(* Logix 5000 project; controller Savage_Saw vendor 1 type 14 code 154 rev 37.11; software revision 37.01; part 2 of 3 *)
(* tags used below, declared in another part *)
   AnyJogRise : BOOL;
   AnyJogStorage : BOOL;
   iAxis : DINT;
   ManualSpinCCW : BOOL;
   ManualSpinCW : BOOL;
   spinActive : BOOL;
   spinDemand : BOOL;
   timerSpinDownCCW : TIMER;
   timerSpinDownCW : TIMER;
   Auto : BOOL;
   AutoCutCancel : BOOL;
   AutoCutCancelFall : BOOL;
   AutoCutCancelOSF : BOOL;
   AutoCutReq : BOOL;
   AutoCutStartONS : BOOL;
   AutoCutStateChange : BOOL;
   AutoSpinCCW : BOOL;
   AutoSpinCW : BOOL;
   Axis : AxisData[3];
   AxisX_Gauge : ALIAS FOR Axis[0];
   AxisY_Traverse : ALIAS FOR Axis[1];
   AxisZ_RaiseLower : ALIAS FOR Axis[2];
   BladeChange10 : BOOL;
   BladeChange10ONS : BOOL;
   BladeChange20 : BOOL;
   BladeChange20ONS : BOOL;
   BladeChangeDone : BOOL;
   BladeChangeStartONS : BOOL;
   BladeChangeStateChange : BOOL;
   BladeMeasure10ONS : BOOL;
   BladeMeasure10StopAll : BOOL;
   BladeMeasure15ClearZero : BOOL;
   BladeMeasure20ONS : BOOL;
   BladeMeasure20Retract : BOOL;
   BladeMeasure30ONS : BOOL;
   BladeMeasure30Traverse : BOOL;
   BladeMeasure40Lower : BOOL;
   BladeMeasure40ONS : BOOL;
   BladeMeasure50ONS : BOOL;
   BladeMeasure50Stop : BOOL;
   BladeMeasure55ONS : BOOL;
   BladeMeasure55Raise : BOOL;
   BladeMeasure60ONS : BOOL;
   BladeMeasure60Stop : BOOL;
   BladeMeasure65Measure : BOOL;
   BladeMeasure65ONS : BOOL;
   BladeMeasure70Calc : BOOL;
   BladeMeasure70ONS : BOOL;
   BladeMeasure75ONS : BOOL;
   BladeMeasure75PartRef : BOOL;
   BladeMeasure80ONS : BOOL;
   BladeMeasure80Return : BOOL;
   BladeMeasureStartONS : BOOL;
   BladeMeasureStateChange : BOOL;
   BladeRadius : REAL;
   BladeRadiusKnown : BOOL;
   BuildDone : BOOL;
   CutEndPosition : REAL;
   CutForward : BOOL;
   CutOnReturn : BOOL;
   CutStartPosition : REAL;
   Fault : BOOL;
   FaultOSR : BOOL;
   FaultRise : BOOL;
   HydReady : BOOL;
   inPe01BladeDetect : ALIAS FOR Local:1:I.Data.7;
   inSR1SafetyRelay : ALIAS FOR Local:1:I.Data.0;
   MC_Reset : ALIAS FOR RMC:O2.Data[3].0;
   NorthZero : BOOL;
   Pass : Pass[21];
   PastPart : REAL;
   RaiseLowerVelocityHome : REAL;
   RaiseLowerVelocityMax : REAL;
   RemainDepth : REAL;
   RpmTarget : REAL;
   RpmTarget105Pct : REAL;
   SafetyRelayAutoReset : BOOL;
   SpinCCWActive : BOOL;
   SpinCCWDemand : BOOL;
   SpinCWActive : BOOL;
   SpinCWDemand : BOOL;
   SpinDemandFall : BOOL;
   SpindlePressure : REAL;
   SpindleRPM : REAL;
   SpindleRPMAtTarget : BOOL;
   SpindleStall : BOOL;
   SpindleStallPressure : REAL;
   SpindleStallRPM : REAL;
   State : DINT;
   State200Build : BOOL;
   State200ONS : BOOL;
   State205 : BOOL;
   State205ONS : BOOL;
   State207ONS : BOOL;
   State207TraverseInitial : BOOL;
   State210Direction : BOOL;
   State210ONS : BOOL;
   State220ONS : BOOL;
   State220TraverseToStart : BOOL;
   State230StartSaw : BOOL;
   State240 : BOOL;
   State240ONS : BOOL;
   State250CheckRPM : BOOL;
   State250ONS : BOOL;
   State260Cut : BOOL;
   State260ONS : BOOL;
   State280 : BOOL;
   State280ONS : BOOL;
   State285BladeMeasure : BOOL;
   State290ONS : BOOL;
   State290RaiseBlade : BOOL;
   State299 : BOOL;
   StepCount : DINT;
   tbA1JogIn : BOOL;
   tbA1JogOut : BOOL;
   tbA2JogMinus : BOOL;
   tbA2JogPlus : BOOL;
   tbA3JogMinus : BOOL;
   tbA3JogPlus : BOOL;
   tbBladeChange : BOOL;
   tbBladeMeasure : BOOL;
   tbCCW : BOOL;
   tbCoolant : BOOL;
   tbCW : BOOL;
   tbHome : BOOL;
   tbNorthRef : BOOL;
   tbSouthRef : BOOL;
   timerAxisZ_RaiseLowerClearZero : TIMER;
   timerSpindleStall : TIMER;
   timerState250CheckRPM : TIMER;
   TraverseRange : REAL;
   TraverseVelocityHome : REAL;
   TraverseVelocityMax : REAL;
   ValidData : BOOL;
   Width : REAL;
   X_AutoCut : BOOL;
   X_BladeChange : BOOL;
   X_BladeMeasure : BOOL;
   X_Fault : BOOL;
   X_Homing : BOOL;
   X_Manual : BOOL;
   X_Off : BOOL;
   X_State : DINT;
(* MainProgram, continued *)

ROUTINE RMC   (* ladder *)
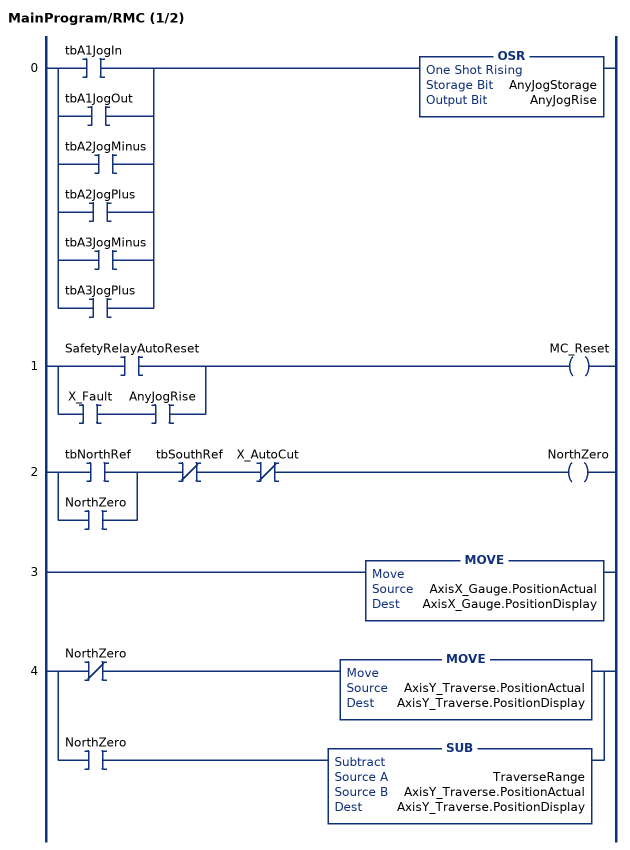
   0: [XIC(tbA1JogIn) ,XIC(tbA1JogOut) ,XIC(tbA2JogMinus) ,XIC(tbA2JogPlus) ,XIC(tbA3JogMinus) ,XIC(tbA3JogPlus) ]OSR(AnyJogStorage,AnyJogRise);
   1: [XIC(SafetyRelayAutoReset) ,XIC(X_Fault) XIC(AnyJogRise) ]OTE(MC_Reset);
   2: [XIC(tbNorthRef) ,XIC(NorthZero) ]XIO(tbSouthRef)XIO(X_AutoCut)OTE(NorthZero);
   3: MOVE(AxisX_Gauge.PositionActual,AxisX_Gauge.PositionDisplay);
   4: [XIO(NorthZero) MOVE(AxisY_Traverse.PositionActual,AxisY_Traverse.PositionDisplay) ,XIC(NorthZero) SUB(TraverseRange,AxisY_Traverse.PositionActual,AxisY_Traverse.PositionDisplay) ];
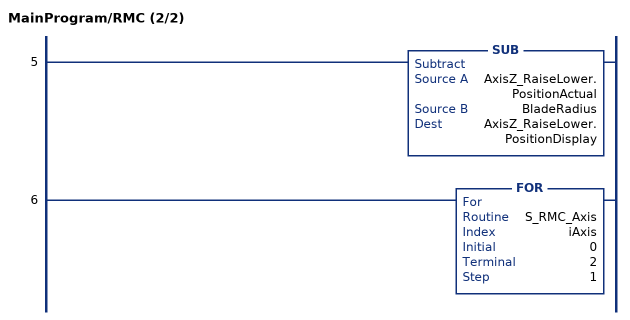
   5: SUB(AxisZ_RaiseLower.PositionActual,BladeRadius,AxisZ_RaiseLower.PositionDisplay);
   6: FOR(S_RMC_Axis,iAxis,0,2,1);
END_ROUTINE

ROUTINE S_RMC_Axis   (* ladder *)
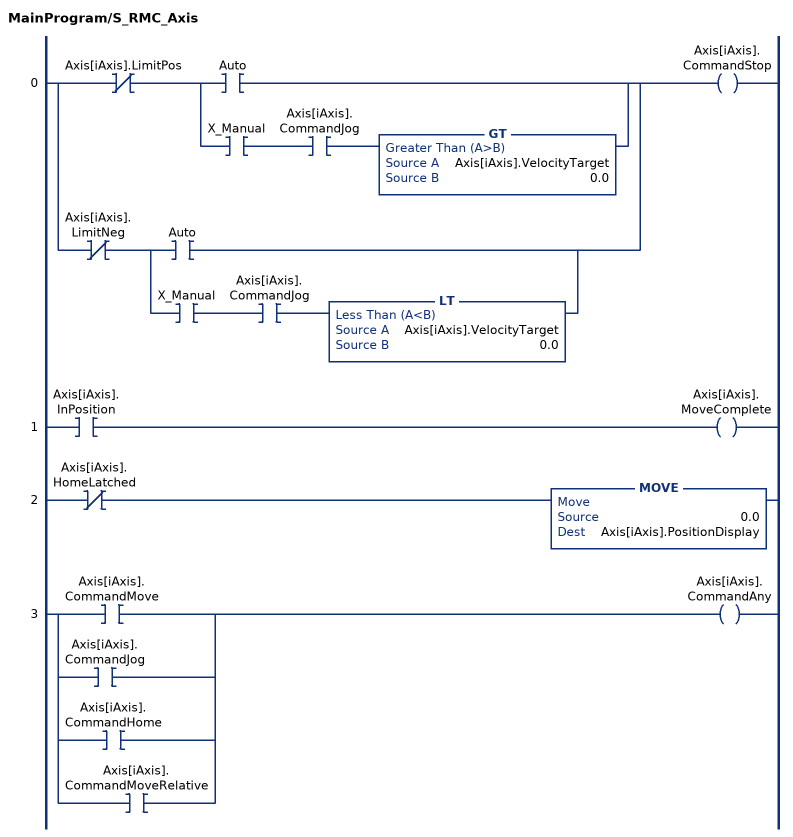
   0: [XIO(Axis[iAxis].LimitPos) [XIC(Auto) ,XIC(X_Manual) XIC(Axis[iAxis].CommandJog) GT(Axis[iAxis].VelocityTarget,0.0) ] ,XIO(Axis[iAxis].LimitNeg) [XIC(Auto) ,XIC(X_Manual) XIC(Axis[iAxis].CommandJog) LT(Axis[iAxis].VelocityTarget,0.0) ] ]OTE(Axis[iAxis].CommandStop);
   1: XIC(Axis[iAxis].InPosition)OTE(Axis[iAxis].MoveComplete);
   2: XIO(Axis[iAxis].HomeLatched)MOVE(0.0,Axis[iAxis].PositionDisplay);
   3: [XIC(Axis[iAxis].CommandMove) ,XIC(Axis[iAxis].CommandJog) ,XIC(Axis[iAxis].CommandHome) ,XIC(Axis[iAxis].CommandMoveRelative) ]OTE(Axis[iAxis].CommandAny);
END_ROUTINE

ROUTINE S_Stop_Axis   (* ladder *)
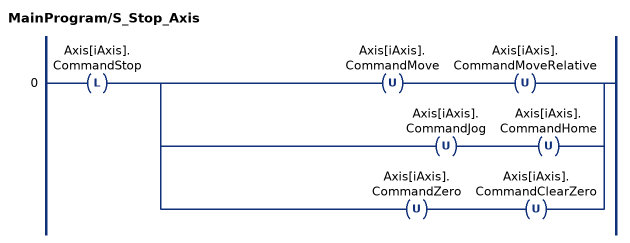
   0: OTL(Axis[iAxis].CommandStop)[OTU(Axis[iAxis].CommandMove) OTU(Axis[iAxis].CommandMoveRelative) ,OTU(Axis[iAxis].CommandJog) OTU(Axis[iAxis].CommandHome) ,OTU(Axis[iAxis].CommandZero) OTU(Axis[iAxis].CommandClearZero) ];
END_ROUTINE

ROUTINE Spindle   (* ladder *)
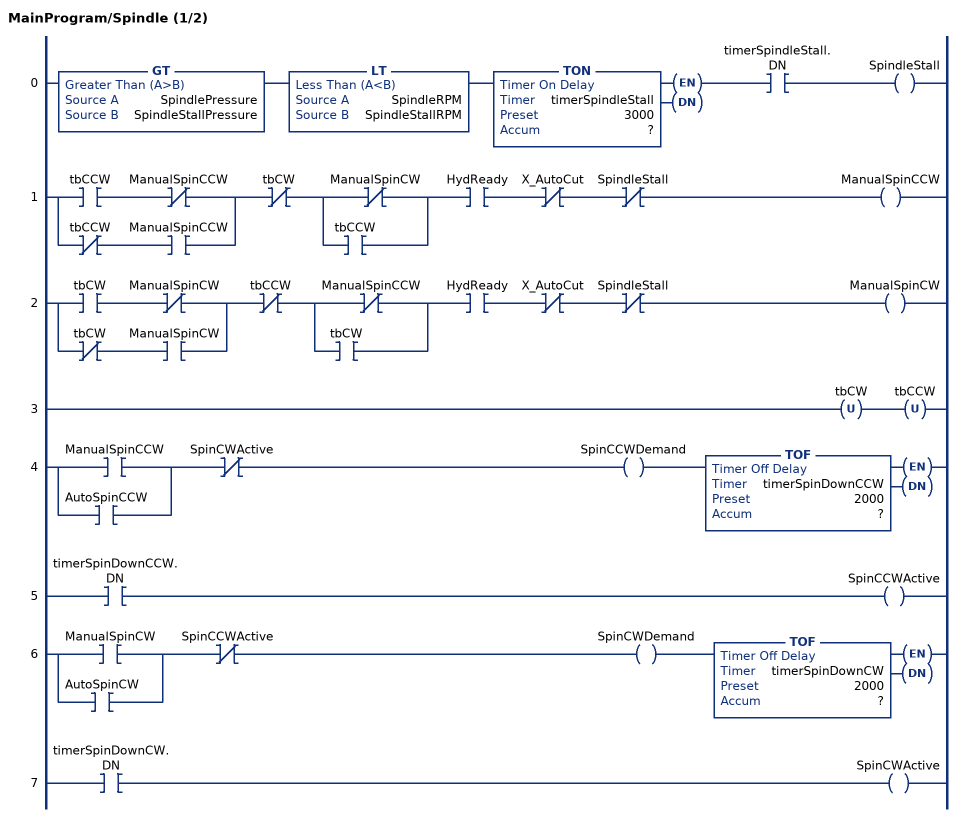
   0: GT(SpindlePressure,SpindleStallPressure)LT(SpindleRPM,SpindleStallRPM)TON(timerSpindleStall,?,?)XIC(timerSpindleStall.DN)OTE(SpindleStall);
   1: [XIC(tbCCW) XIO(ManualSpinCCW) ,XIO(tbCCW) XIC(ManualSpinCCW) ]XIO(tbCW)[XIO(ManualSpinCW) ,XIC(tbCCW) ]XIC(HydReady)XIO(X_AutoCut)XIO(SpindleStall)OTE(ManualSpinCCW);
   2: [XIC(tbCW) XIO(ManualSpinCW) ,XIO(tbCW) XIC(ManualSpinCW) ]XIO(tbCCW)[XIO(ManualSpinCCW) ,XIC(tbCW) ]XIC(HydReady)XIO(X_AutoCut)XIO(SpindleStall)OTE(ManualSpinCW);
   3: OTU(tbCW)OTU(tbCCW);
   4: [XIC(ManualSpinCCW) ,XIC(AutoSpinCCW) ]XIO(SpinCWActive)OTE(SpinCCWDemand)TOF(timerSpinDownCCW,?,?);
   5: XIC(timerSpinDownCCW.DN)OTE(SpinCCWActive);
   6: [XIC(ManualSpinCW) ,XIC(AutoSpinCW) ]XIO(SpinCCWActive)OTE(SpinCWDemand)TOF(timerSpinDownCW,?,?);
   7: XIC(timerSpinDownCW.DN)OTE(SpinCWActive);
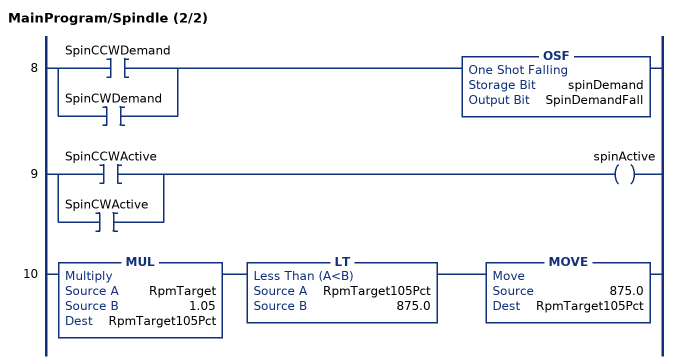
   8: [XIC(SpinCCWDemand) ,XIC(SpinCWDemand) ]OSF(spinDemand,SpinDemandFall);
   9: [XIC(SpinCCWActive) ,XIC(SpinCWActive) ]OTE(spinActive);
   10: MUL(RpmTarget,1.05,RpmTarget105Pct)LT(RpmTarget105Pct,875.0)MOVE(875.0,RpmTarget105Pct);
END_ROUTINE

ROUTINE State   (* ladder *)
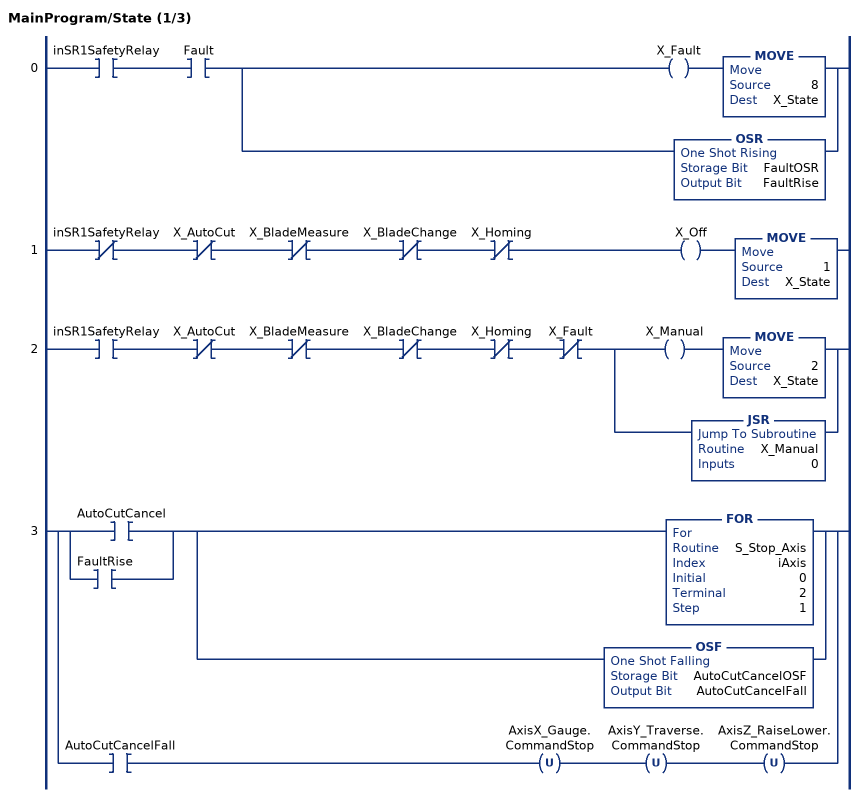
   0: XIC(inSR1SafetyRelay)XIC(Fault)[OTE(X_Fault) MOVE(8,X_State) ,OSR(FaultOSR,FaultRise) ];
   1: XIO(inSR1SafetyRelay)XIO(X_AutoCut)XIO(X_BladeMeasure)XIO(X_BladeChange)XIO(X_Homing)OTE(X_Off)MOVE(1,X_State);
   2: XIC(inSR1SafetyRelay)XIO(X_AutoCut)XIO(X_BladeMeasure)XIO(X_BladeChange)XIO(X_Homing)XIO(X_Fault)[OTE(X_Manual) MOVE(2,X_State) ,JSR(X_Manual,0) ];
   3: [[XIC(AutoCutCancel) ,XIC(FaultRise) ] [FOR(S_Stop_Axis,iAxis,0,2,1) ,OSF(AutoCutCancelOSF,AutoCutCancelFall) ] ,XIC(AutoCutCancelFall) OTU(AxisX_Gauge.CommandStop) OTU(AxisY_Traverse.CommandStop) OTU(AxisZ_RaiseLower.CommandStop) ];
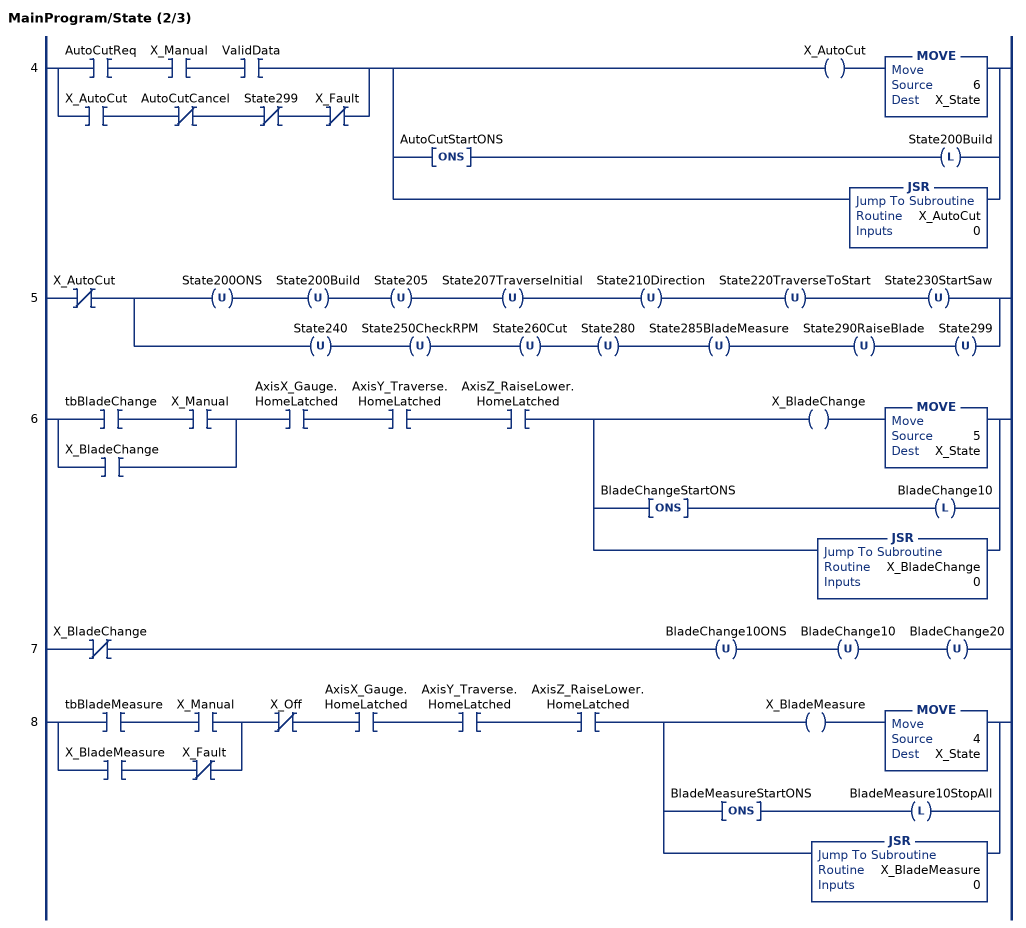
   4: [XIC(AutoCutReq) XIC(X_Manual) XIC(ValidData) ,XIC(X_AutoCut) XIO(AutoCutCancel) XIO(State299) XIO(X_Fault) ][OTE(X_AutoCut) MOVE(6,X_State) ,ONS(AutoCutStartONS) OTL(State200Build) ,JSR(X_AutoCut,0) ];
   5: XIO(X_AutoCut)[OTU(State200ONS) OTU(State200Build) OTU(State205) OTU(State207TraverseInitial) OTU(State210Direction) OTU(State220TraverseToStart) OTU(State230StartSaw) ,OTU(State240) OTU(State250CheckRPM) OTU(State260Cut) OTU(State280) OTU(State285BladeMeasure) OTU(State290RaiseBlade) OTU(State299) ];
   6: [XIC(tbBladeChange) XIC(X_Manual) ,XIC(X_BladeChange) ]XIC(AxisX_Gauge.HomeLatched)XIC(AxisY_Traverse.HomeLatched)XIC(AxisZ_RaiseLower.HomeLatched)[OTE(X_BladeChange) MOVE(5,X_State) ,ONS(BladeChangeStartONS) OTL(BladeChange10) ,JSR(X_BladeChange,0) ];
   7: XIO(X_BladeChange)OTU(BladeChange10ONS)OTU(BladeChange10)OTU(BladeChange20);
   8: [XIC(tbBladeMeasure) XIC(X_Manual) ,XIC(X_BladeMeasure) XIO(X_Fault) ]XIO(X_Off)XIC(AxisX_Gauge.HomeLatched)XIC(AxisY_Traverse.HomeLatched)XIC(AxisZ_RaiseLower.HomeLatched)[OTE(X_BladeMeasure) MOVE(4,X_State) ,ONS(BladeMeasureStartONS) OTL(BladeMeasure10StopAll) ,JSR(X_BladeMeasure,0) ];
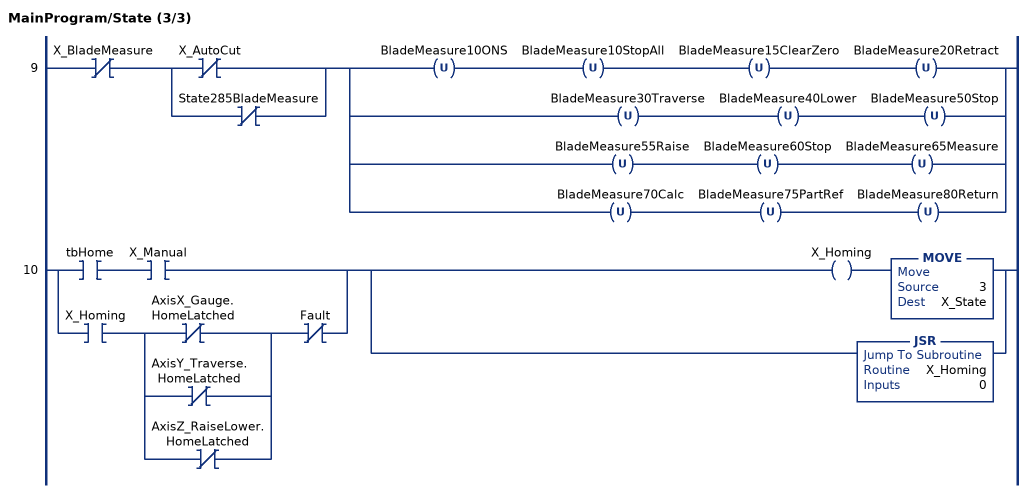
   9: XIO(X_BladeMeasure)[XIO(X_AutoCut) ,XIO(State285BladeMeasure) ][OTU(BladeMeasure10ONS) OTU(BladeMeasure10StopAll) OTU(BladeMeasure15ClearZero) OTU(BladeMeasure20Retract) ,OTU(BladeMeasure30Traverse) OTU(BladeMeasure40Lower) OTU(BladeMeasure50Stop) ,OTU(BladeMeasure55Raise) OTU(BladeMeasure60Stop) OTU(BladeMeasure65Measure) ,OTU(BladeMeasure70Calc) OTU(BladeMeasure75PartRef) OTU(BladeMeasure80Return) ];
   10: [XIC(tbHome) XIC(X_Manual) ,XIC(X_Homing) [XIO(AxisX_Gauge.HomeLatched) ,XIO(AxisY_Traverse.HomeLatched) ,XIO(AxisZ_RaiseLower.HomeLatched) ] XIO(Fault) ][OTE(X_Homing) MOVE(3,X_State) ,JSR(X_Homing,0) ];
END_ROUTINE

ROUTINE X_AutoCut   (* ladder *)
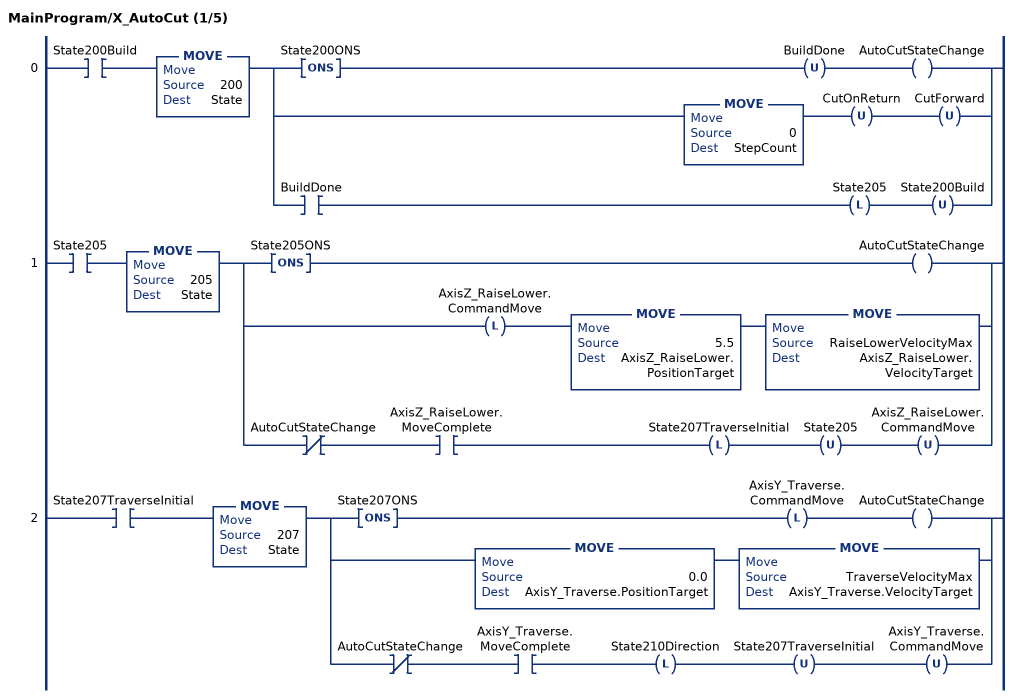
   0: XIC(State200Build)MOVE(200,State)[ONS(State200ONS) OTU(BuildDone) OTE(AutoCutStateChange) ,MOVE(0,StepCount) OTU(CutOnReturn) OTU(CutForward) ,XIC(BuildDone) OTL(State205) OTU(State200Build) ];
   1: XIC(State205)MOVE(205,State)[ONS(State205ONS) OTE(AutoCutStateChange) ,OTL(AxisZ_RaiseLower.CommandMove) MOVE(5.5,AxisZ_RaiseLower.PositionTarget) MOVE(RaiseLowerVelocityMax,AxisZ_RaiseLower.VelocityTarget) ,XIO(AutoCutStateChange) XIC(AxisZ_RaiseLower.MoveComplete) OTL(State207TraverseInitial) OTU(State205) OTU(AxisZ_RaiseLower.CommandMove) ];
   2: XIC(State207TraverseInitial)MOVE(207,State)[ONS(State207ONS) OTL(AxisY_Traverse.CommandMove) OTE(AutoCutStateChange) ,MOVE(0.0,AxisY_Traverse.PositionTarget) MOVE(TraverseVelocityMax,AxisY_Traverse.VelocityTarget) ,XIO(AutoCutStateChange) XIC(AxisY_Traverse.MoveComplete) OTL(State210Direction) OTU(State207TraverseInitial) OTU(AxisY_Traverse.CommandMove) ];
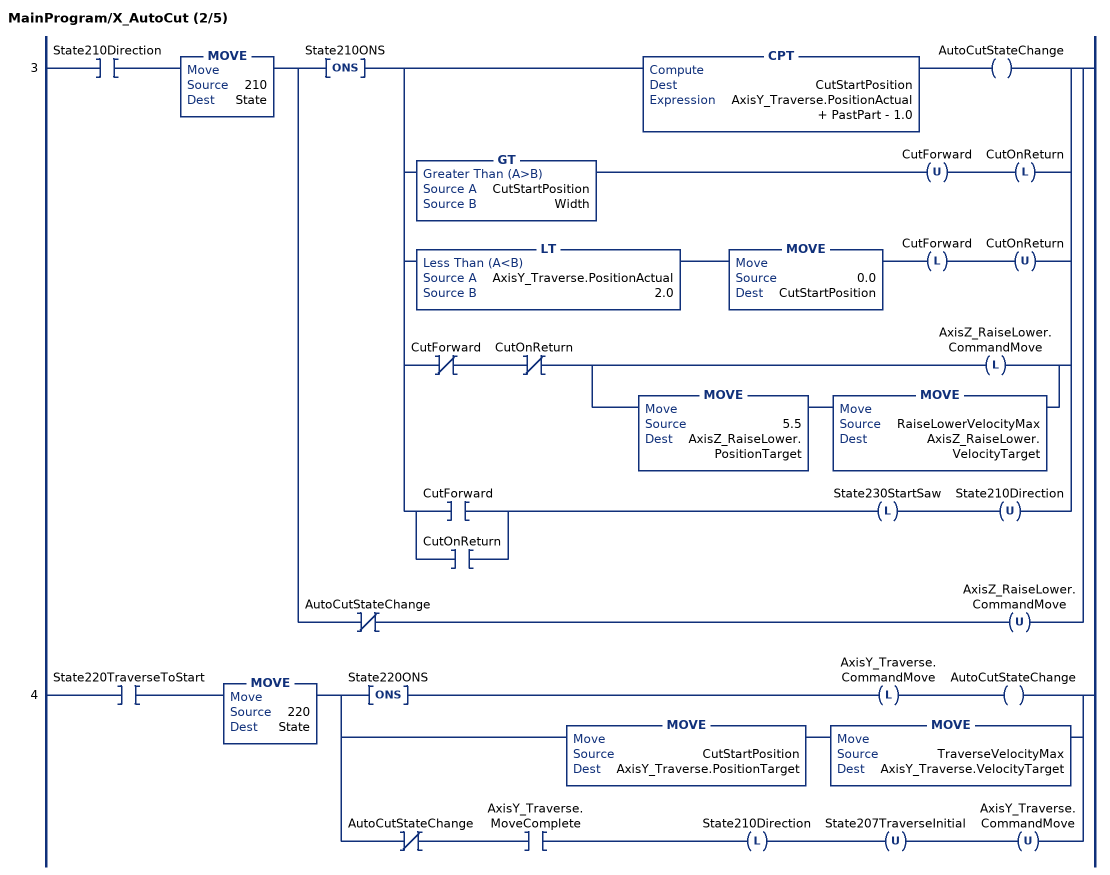
   3: XIC(State210Direction)MOVE(210,State)[ONS(State210ONS) [CPT(CutStartPosition,AxisY_Traverse.PositionActual + PastPart - 1.0) OTE(AutoCutStateChange) ,GT(CutStartPosition,Width) OTU(CutForward) OTL(CutOnReturn) ,LT(AxisY_Traverse.PositionActual,2.0) MOVE(0.0,CutStartPosition) OTL(CutForward) OTU(CutOnReturn) ,XIO(CutForward) XIO(CutOnReturn) [OTL(AxisZ_RaiseLower.CommandMove) ,MOVE(5.5,AxisZ_RaiseLower.PositionTarget) MOVE(RaiseLowerVelocityMax,AxisZ_RaiseLower.VelocityTarget) ] ,[XIC(CutForward) ,XIC(CutOnReturn) ] OTL(State230StartSaw) OTU(State210Direction) ] ,XIO(AutoCutStateChange) OTU(AxisZ_RaiseLower.CommandMove) ];
   4: XIC(State220TraverseToStart)MOVE(220,State)[ONS(State220ONS) OTL(AxisY_Traverse.CommandMove) OTE(AutoCutStateChange) ,MOVE(CutStartPosition,AxisY_Traverse.PositionTarget) MOVE(TraverseVelocityMax,AxisY_Traverse.VelocityTarget) ,XIO(AutoCutStateChange) XIC(AxisY_Traverse.MoveComplete) OTL(State210Direction) OTU(State207TraverseInitial) OTU(AxisY_Traverse.CommandMove) ];
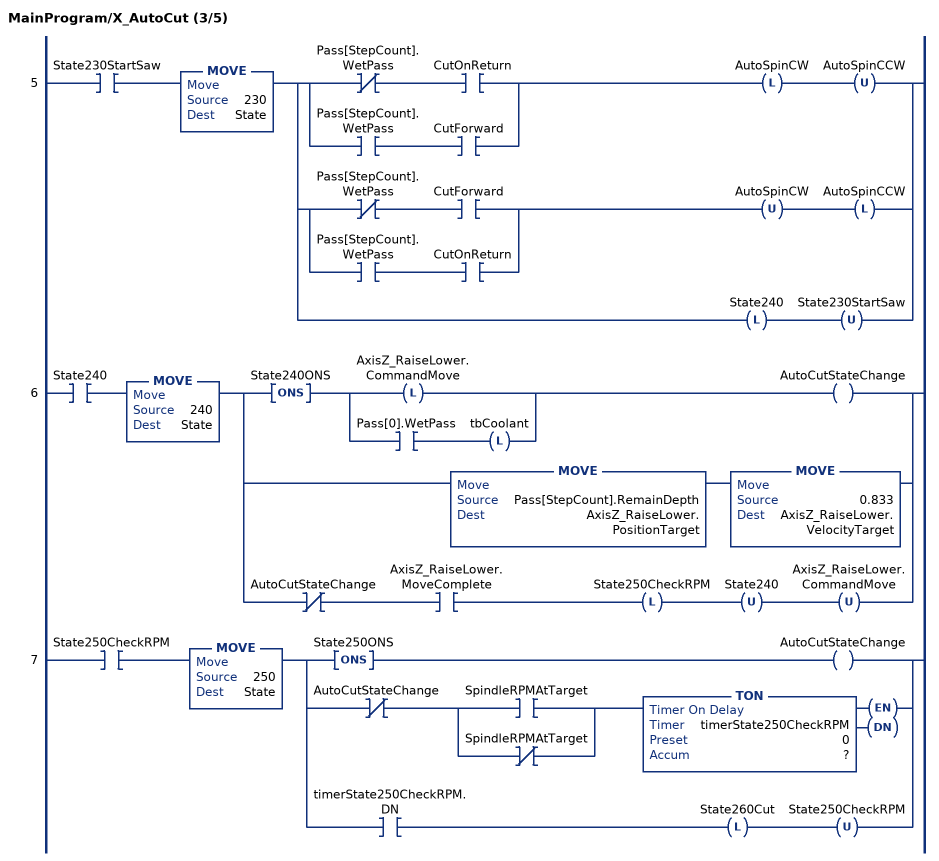
   5: XIC(State230StartSaw)MOVE(230,State)[[XIO(Pass[StepCount].WetPass) XIC(CutOnReturn) ,XIC(Pass[StepCount].WetPass) XIC(CutForward) ] OTL(AutoSpinCW) OTU(AutoSpinCCW) ,[XIO(Pass[StepCount].WetPass) XIC(CutForward) ,XIC(Pass[StepCount].WetPass) XIC(CutOnReturn) ] OTU(AutoSpinCW) OTL(AutoSpinCCW) ,OTL(State240) OTU(State230StartSaw) ];
   6: XIC(State240)MOVE(240,State)[ONS(State240ONS) [OTL(AxisZ_RaiseLower.CommandMove) ,XIC(Pass[0].WetPass) OTL(tbCoolant) ] OTE(AutoCutStateChange) ,MOVE(Pass[StepCount].RemainDepth,AxisZ_RaiseLower.PositionTarget) MOVE(0.833,AxisZ_RaiseLower.VelocityTarget) ,XIO(AutoCutStateChange) XIC(AxisZ_RaiseLower.MoveComplete) OTL(State250CheckRPM) OTU(State240) OTU(AxisZ_RaiseLower.CommandMove) ];
   7: XIC(State250CheckRPM)MOVE(250,State)[ONS(State250ONS) OTE(AutoCutStateChange) ,XIO(AutoCutStateChange) [XIC(SpindleRPMAtTarget) ,XIO(SpindleRPMAtTarget) ] TON(timerState250CheckRPM,?,?) ,XIC(timerState250CheckRPM.DN) OTL(State260Cut) OTU(State250CheckRPM) ];
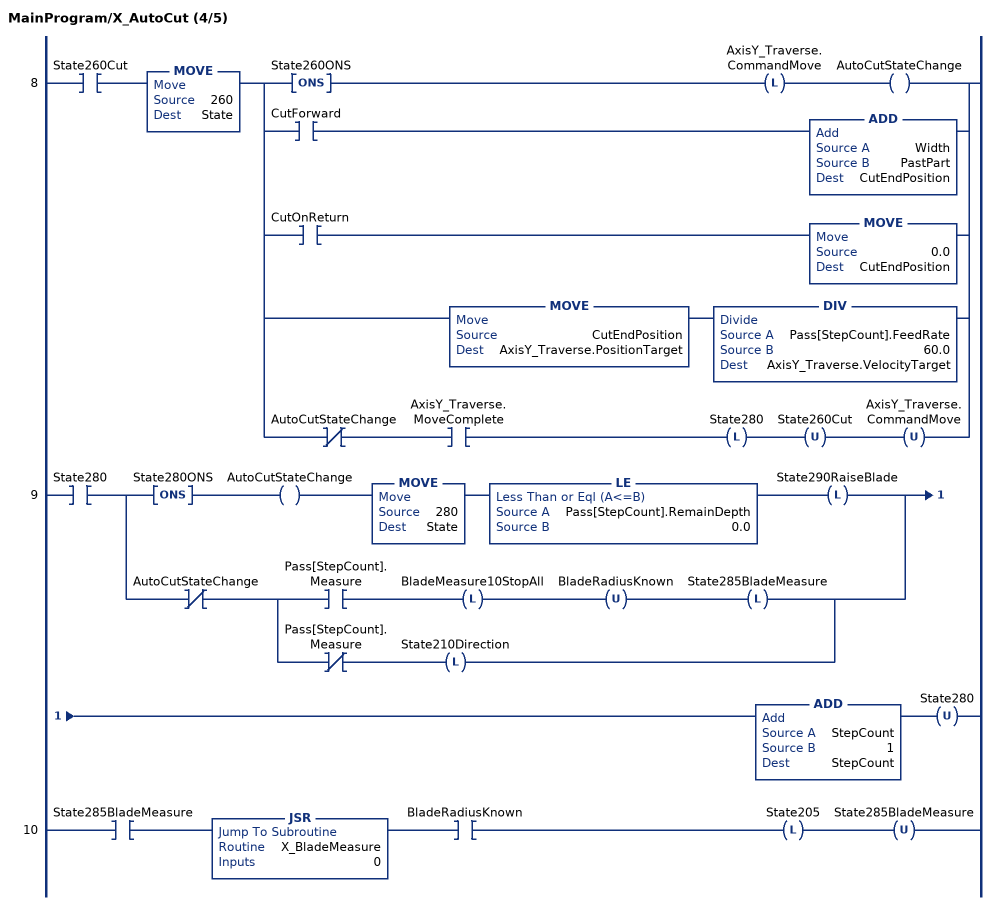
   8: XIC(State260Cut)MOVE(260,State)[ONS(State260ONS) OTL(AxisY_Traverse.CommandMove) OTE(AutoCutStateChange) ,XIC(CutForward) ADD(Width,PastPart,CutEndPosition) ,XIC(CutOnReturn) MOVE(0.0,CutEndPosition) ,MOVE(CutEndPosition,AxisY_Traverse.PositionTarget) DIV(Pass[StepCount].FeedRate,60.0,AxisY_Traverse.VelocityTarget) ,XIO(AutoCutStateChange) XIC(AxisY_Traverse.MoveComplete) OTL(State280) OTU(State260Cut) OTU(AxisY_Traverse.CommandMove) ];
   9: XIC(State280)[ONS(State280ONS) OTE(AutoCutStateChange) MOVE(280,State) LE(Pass[StepCount].RemainDepth,0.0) OTL(State290RaiseBlade) ,XIO(AutoCutStateChange) [XIC(Pass[StepCount].Measure) OTL(BladeMeasure10StopAll) OTU(BladeRadiusKnown) OTL(State285BladeMeasure) ,XIO(Pass[StepCount].Measure) OTL(State210Direction) ] ]ADD(StepCount,1,StepCount)OTU(State280);
   10: XIC(State285BladeMeasure)JSR(X_BladeMeasure,0)XIC(BladeRadiusKnown)OTL(State205)OTU(State285BladeMeasure);
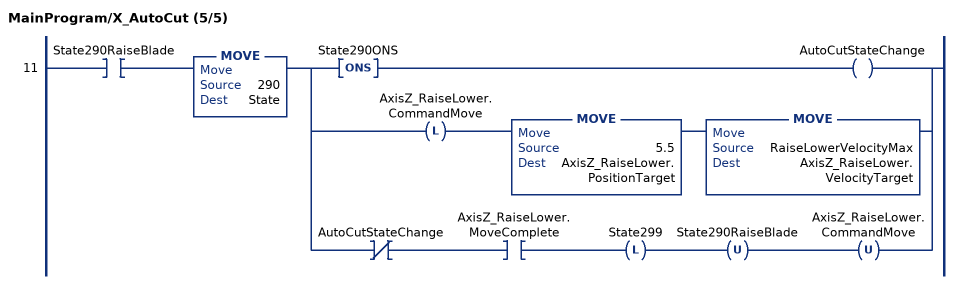
   11: XIC(State290RaiseBlade)MOVE(290,State)[ONS(State290ONS) OTE(AutoCutStateChange) ,OTL(AxisZ_RaiseLower.CommandMove) MOVE(5.5,AxisZ_RaiseLower.PositionTarget) MOVE(RaiseLowerVelocityMax,AxisZ_RaiseLower.VelocityTarget) ,XIO(AutoCutStateChange) XIC(AxisZ_RaiseLower.MoveComplete) OTL(State299) OTU(State290RaiseBlade) OTU(AxisZ_RaiseLower.CommandMove) ];
END_ROUTINE

ROUTINE X_BladeChange   (* ladder *)
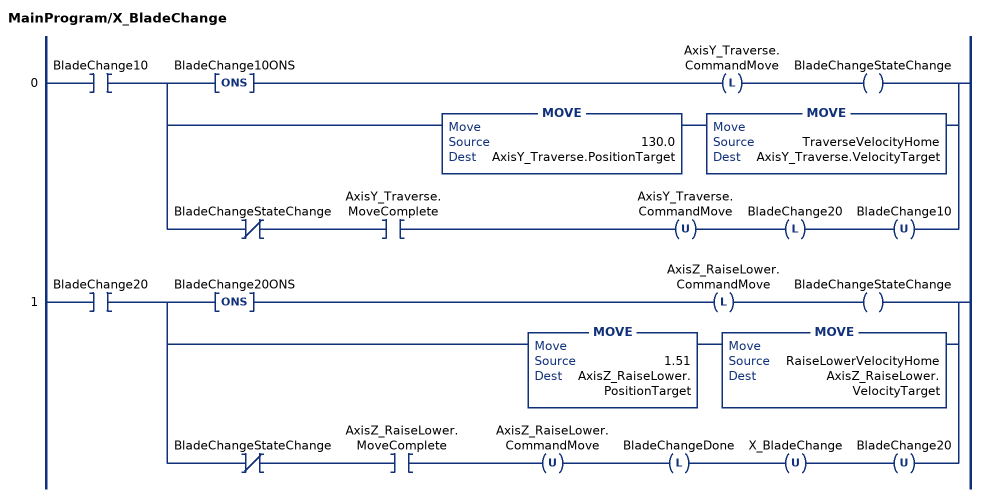
   0: XIC(BladeChange10)[ONS(BladeChange10ONS) OTL(AxisY_Traverse.CommandMove) OTE(BladeChangeStateChange) ,MOVE(130.0,AxisY_Traverse.PositionTarget) MOVE(TraverseVelocityHome,AxisY_Traverse.VelocityTarget) ,XIO(BladeChangeStateChange) XIC(AxisY_Traverse.MoveComplete) OTU(AxisY_Traverse.CommandMove) OTL(BladeChange20) OTU(BladeChange10) ];
   1: XIC(BladeChange20)[ONS(BladeChange20ONS) OTL(AxisZ_RaiseLower.CommandMove) OTE(BladeChangeStateChange) ,MOVE(1.51,AxisZ_RaiseLower.PositionTarget) MOVE(RaiseLowerVelocityHome,AxisZ_RaiseLower.VelocityTarget) ,XIO(BladeChangeStateChange) XIC(AxisZ_RaiseLower.MoveComplete) OTU(AxisZ_RaiseLower.CommandMove) OTL(BladeChangeDone) OTU(X_BladeChange) OTU(BladeChange20) ];
END_ROUTINE

ROUTINE X_BladeMeasure   (* ladder *)
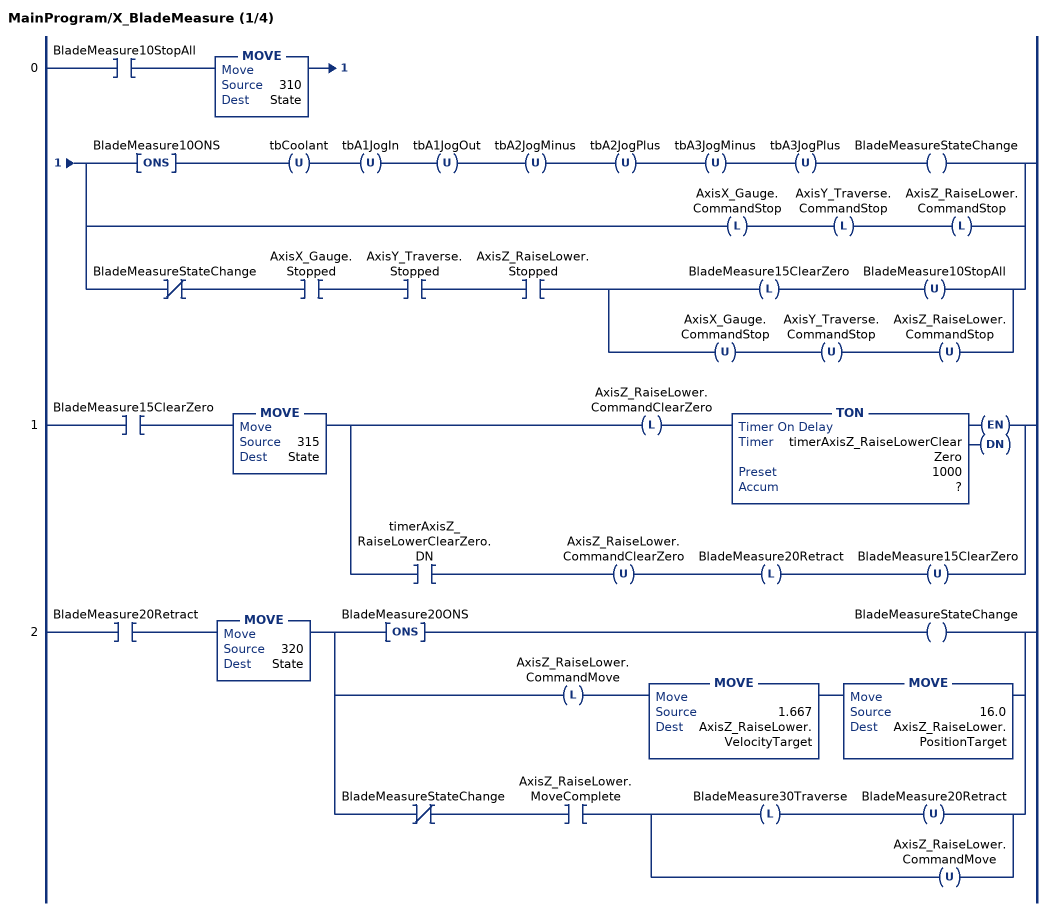
   0: XIC(BladeMeasure10StopAll)MOVE(310,State)[ONS(BladeMeasure10ONS) OTU(tbCoolant) OTU(tbA1JogIn) OTU(tbA1JogOut) OTU(tbA2JogMinus) OTU(tbA2JogPlus) OTU(tbA3JogMinus) OTU(tbA3JogPlus) OTE(BladeMeasureStateChange) ,OTL(AxisX_Gauge.CommandStop) OTL(AxisY_Traverse.CommandStop) OTL(AxisZ_RaiseLower.CommandStop) ,XIO(BladeMeasureStateChange) XIC(AxisX_Gauge.Stopped) XIC(AxisY_Traverse.Stopped) XIC(AxisZ_RaiseLower.Stopped) [OTL(BladeMeasure15ClearZero) OTU(BladeMeasure10StopAll) ,OTU(AxisX_Gauge.CommandStop) OTU(AxisY_Traverse.CommandStop) OTU(AxisZ_RaiseLower.CommandStop) ] ];
   1: XIC(BladeMeasure15ClearZero)MOVE(315,State)[OTL(AxisZ_RaiseLower.CommandClearZero) TON(timerAxisZ_RaiseLowerClearZero,?,?) ,XIC(timerAxisZ_RaiseLowerClearZero.DN) OTU(AxisZ_RaiseLower.CommandClearZero) OTL(BladeMeasure20Retract) OTU(BladeMeasure15ClearZero) ];
   2: XIC(BladeMeasure20Retract)MOVE(320,State)[ONS(BladeMeasure20ONS) OTE(BladeMeasureStateChange) ,OTL(AxisZ_RaiseLower.CommandMove) MOVE(1.667,AxisZ_RaiseLower.VelocityTarget) MOVE(16.0,AxisZ_RaiseLower.PositionTarget) ,XIO(BladeMeasureStateChange) XIC(AxisZ_RaiseLower.MoveComplete) [OTL(BladeMeasure30Traverse) OTU(BladeMeasure20Retract) ,OTU(AxisZ_RaiseLower.CommandMove) ] ];
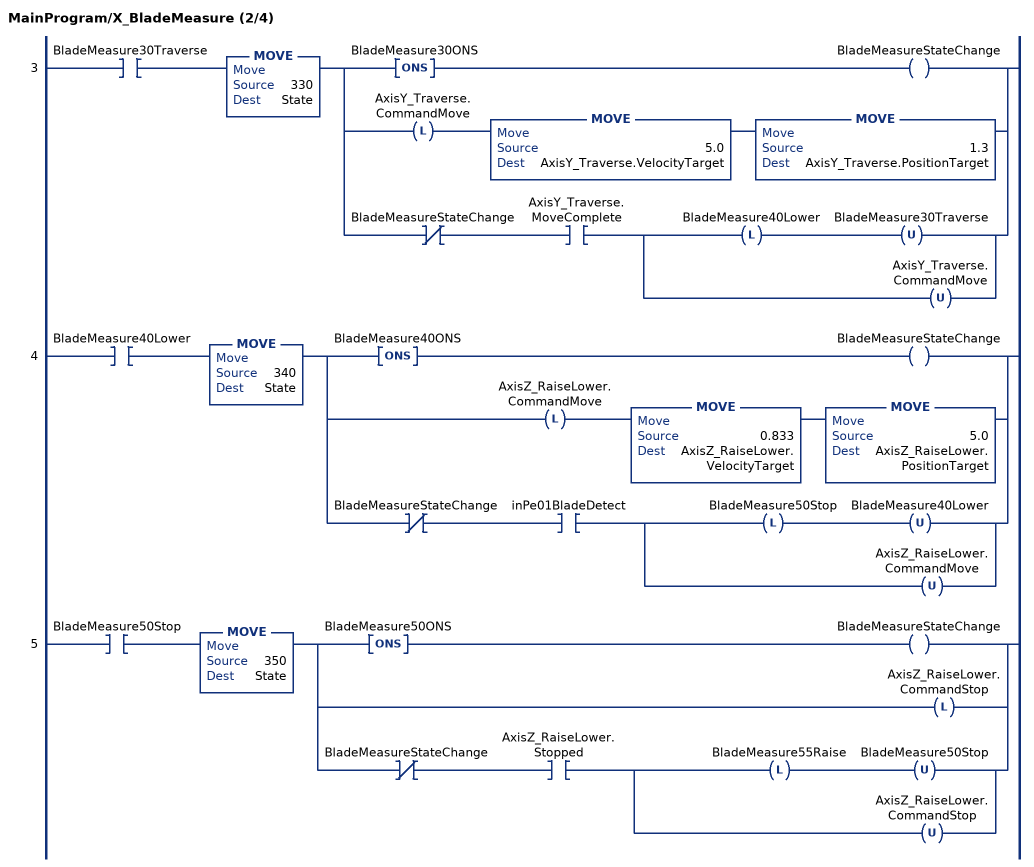
   3: XIC(BladeMeasure30Traverse)MOVE(330,State)[ONS(BladeMeasure30ONS) OTE(BladeMeasureStateChange) ,OTL(AxisY_Traverse.CommandMove) MOVE(5.0,AxisY_Traverse.VelocityTarget) MOVE(1.3,AxisY_Traverse.PositionTarget) ,XIO(BladeMeasureStateChange) XIC(AxisY_Traverse.MoveComplete) [OTL(BladeMeasure40Lower) OTU(BladeMeasure30Traverse) ,OTU(AxisY_Traverse.CommandMove) ] ];
   4: XIC(BladeMeasure40Lower)MOVE(340,State)[ONS(BladeMeasure40ONS) OTE(BladeMeasureStateChange) ,OTL(AxisZ_RaiseLower.CommandMove) MOVE(0.833,AxisZ_RaiseLower.VelocityTarget) MOVE(5.0,AxisZ_RaiseLower.PositionTarget) ,XIO(BladeMeasureStateChange) XIC(inPe01BladeDetect) [OTL(BladeMeasure50Stop) OTU(BladeMeasure40Lower) ,OTU(AxisZ_RaiseLower.CommandMove) ] ];
   5: XIC(BladeMeasure50Stop)MOVE(350,State)[ONS(BladeMeasure50ONS) OTE(BladeMeasureStateChange) ,OTL(AxisZ_RaiseLower.CommandStop) ,XIO(BladeMeasureStateChange) XIC(AxisZ_RaiseLower.Stopped) [OTL(BladeMeasure55Raise) OTU(BladeMeasure50Stop) ,OTU(AxisZ_RaiseLower.CommandStop) ] ];
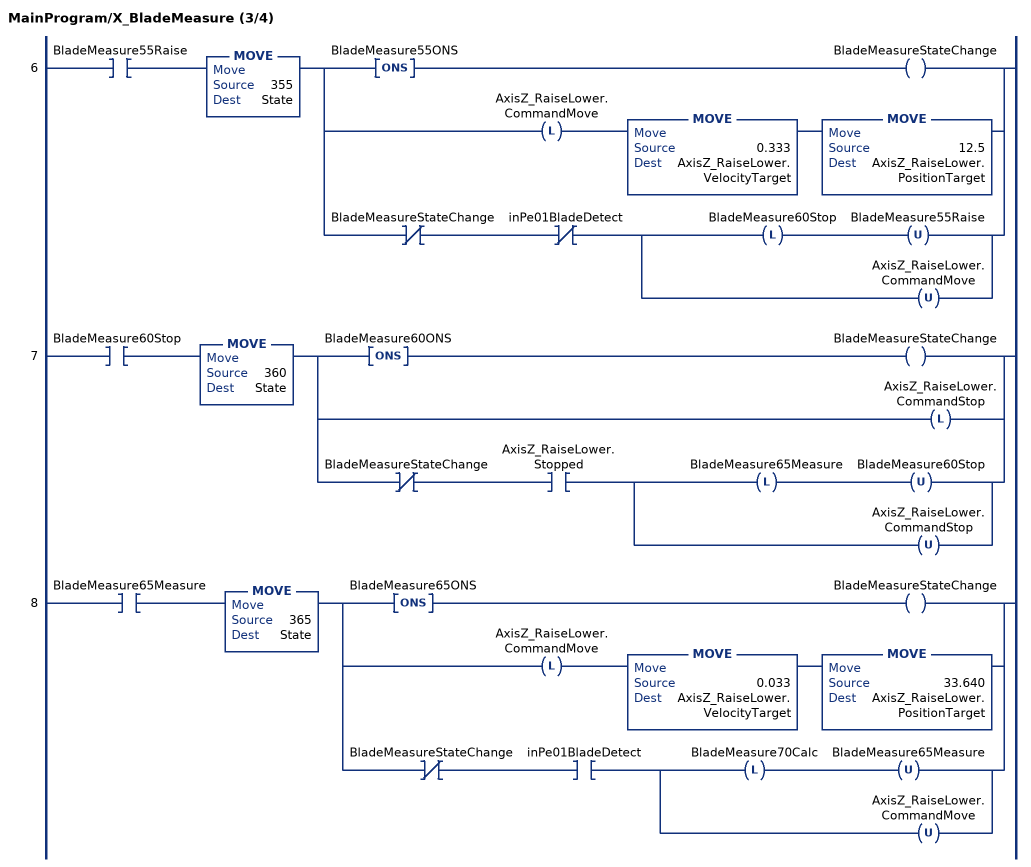
   6: XIC(BladeMeasure55Raise)MOVE(355,State)[ONS(BladeMeasure55ONS) OTE(BladeMeasureStateChange) ,OTL(AxisZ_RaiseLower.CommandMove) MOVE(0.333,AxisZ_RaiseLower.VelocityTarget) MOVE(12.5,AxisZ_RaiseLower.PositionTarget) ,XIO(BladeMeasureStateChange) XIO(inPe01BladeDetect) [OTL(BladeMeasure60Stop) OTU(BladeMeasure55Raise) ,OTU(AxisZ_RaiseLower.CommandMove) ] ];
   7: XIC(BladeMeasure60Stop)MOVE(360,State)[ONS(BladeMeasure60ONS) OTE(BladeMeasureStateChange) ,OTL(AxisZ_RaiseLower.CommandStop) ,XIO(BladeMeasureStateChange) XIC(AxisZ_RaiseLower.Stopped) [OTL(BladeMeasure65Measure) OTU(BladeMeasure60Stop) ,OTU(AxisZ_RaiseLower.CommandStop) ] ];
   8: XIC(BladeMeasure65Measure)MOVE(365,State)[ONS(BladeMeasure65ONS) OTE(BladeMeasureStateChange) ,OTL(AxisZ_RaiseLower.CommandMove) MOVE(0.033,AxisZ_RaiseLower.VelocityTarget) MOVE(33.640,AxisZ_RaiseLower.PositionTarget) ,XIO(BladeMeasureStateChange) XIC(inPe01BladeDetect) [OTL(BladeMeasure70Calc) OTU(BladeMeasure65Measure) ,OTU(AxisZ_RaiseLower.CommandMove) ] ];
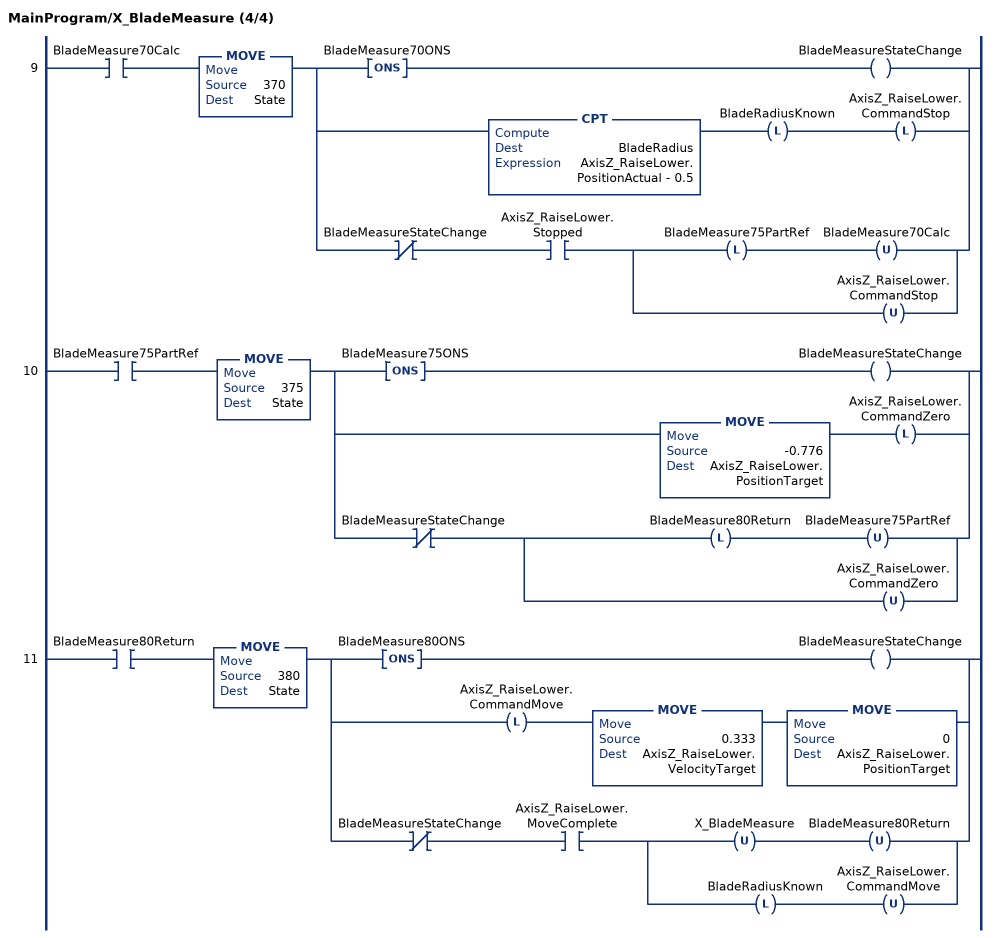
   9: XIC(BladeMeasure70Calc)MOVE(370,State)[ONS(BladeMeasure70ONS) OTE(BladeMeasureStateChange) ,CPT(BladeRadius,AxisZ_RaiseLower.PositionActual - 0.5) OTL(BladeRadiusKnown) OTL(AxisZ_RaiseLower.CommandStop) ,XIO(BladeMeasureStateChange) XIC(AxisZ_RaiseLower.Stopped) [OTL(BladeMeasure75PartRef) OTU(BladeMeasure70Calc) ,OTU(AxisZ_RaiseLower.CommandStop) ] ];
   10: XIC(BladeMeasure75PartRef)MOVE(375,State)[ONS(BladeMeasure75ONS) OTE(BladeMeasureStateChange) ,MOVE(-0.776,AxisZ_RaiseLower.PositionTarget) OTL(AxisZ_RaiseLower.CommandZero) ,XIO(BladeMeasureStateChange) [OTL(BladeMeasure80Return) OTU(BladeMeasure75PartRef) ,OTU(AxisZ_RaiseLower.CommandZero) ] ];
   11: XIC(BladeMeasure80Return)MOVE(380,State)[ONS(BladeMeasure80ONS) OTE(BladeMeasureStateChange) ,OTL(AxisZ_RaiseLower.CommandMove) MOVE(0.333,AxisZ_RaiseLower.VelocityTarget) MOVE(0,AxisZ_RaiseLower.PositionTarget) ,XIO(BladeMeasureStateChange) XIC(AxisZ_RaiseLower.MoveComplete) [OTU(X_BladeMeasure) OTU(BladeMeasure80Return) ,OTL(BladeRadiusKnown) OTU(AxisZ_RaiseLower.CommandMove) ] ];
END_ROUTINE
